Staubli VAL3: onEnterEvent.pgx

program onEnterEvent()
begin
  //
  // NB sEvent is the selected
  // element in the LIST
  //
end
